PROGRAM MAIN
VAR
	bInit 	  : BOOL := FALSE; // flag for initialization
	bTaskDone : BOOL := FALSE;
END_VAR


// Command related
VAR
	fb_CommandProcess : FB_CommandProcess; // Process data from host and transfer data to Cpp
END_VAR
	
// Scope Server
VAR
	fb_GenerateFileSuffixByTime : FB_GenerateFileSuffixByTime; 	// Generate file suffix by system time
	fb_ScopeServer 		  		: FB_ScopeServer; 	  			// Record .svdx file
	bScopeRun 			  		: BOOL := FALSE; 		  		// Flag of starting or stoping scope server
	fb_ExportScopeData 	  		: FB_ExportScopeData;   		// Export recorded data after finishing 
	bExportData    		  		: BOOL := FALSE; 		  		// Flag of exporting data to file
END_VAR

// Initialize and Config load
VAR
	bBufferFilled 	 : BOOL := FALSE; // Flag reflects success or failure of initializing ring buffer
	bMcInfoLoaded 	 : BOOL := FALSE; // Flag reflects success or failure of loading motor info file
	bPanelInfoLoaded : BOOL := FALSE; // Flag reflects success or failure of loading panel info file
	fb_MotorInfoLoad : FB_MotorInfoLoad;
END_VAR

IF (NOT bInit) THEN
	
	bInit := mInitialize();
	
ELSE
	
	mInput();
	
	mOutput();
	
END_IF


// Scope Data Record
fb_ScopeServer(
	bExternalTriggerEvent	:= bScopeRun , 
	sConfigFile				:= GlobalVar.RECORD_CONFIG_PATH, 
	sSaveFile				:= CONCAT(GlobalVar.SAVE_SVDX_PREFIX, fb_GenerateFileSuffixByTime.SAVE_SVDX_SUFFIX));
	
fb_ExportScopeData(
	sNetId					:= '' , 
	bExport					:= bExportData , 
	svd						:= fb_ScopeServer.sSaveFile , 
	target					:= CONCAT(GlobalVar.SAVE_CSV_PREFIX, fb_GenerateFileSuffixByTime.SAVE_CSV_SUFFIX) , 
	config					:= GlobalVar.RECORD_CONFIG_XML_PATH);

METHOD mInitialize : BOOL
// Wait for the following initialization
// Step 1. Host Machine fills command buffer;
// Step 2. Current module finish loading MotionControl xml file;
// Step 3. Current module finish loading Panel xml file;
mInitialize := FALSE;

// Get time to generate suffix of files saved by scope server
fb_GenerateFileSuffixByTime();

// Step 1
IF NOT bBufferFilled THEN
	bBufferFilled := fb_CommandProcess.mInitialize();
END_IF


// Step 2 
IF NOT bMcInfoLoaded THEN
	fb_MotorInfoLoad();
	bMcInfoLoaded := fb_MotorInfoLoad.bExecuteSuccess;
END_IF


// Step 3
IF NOT bPanelInfoLoaded THEN
	bPanelInfoLoaded := TRUE;
END_IF

// Finish all initialization steps.
IF bBufferFilled AND bMcInfoLoaded AND bPanelInfoLoaded THEN
	
	// Start recording data
	bScopeRun := TRUE;
	
	// End initialization
	mInitialize := TRUE;
END_IF
END_METHOD

METHOD mInput : BOOL
VAR_INPUT
END_VAR
// Receive inputs from Hardware and other modules.
END_METHOD

METHOD mOutput : BOOL
VAR_INPUT
END_VAR
// Send outputs to Hardware and other modules.

mOutput := FALSE;

IF fb_CommandProcess.mSendCommand() THEN
	mOutput := TRUE;
ELSE
	// TODO: add judgment on whether the task is finished
	IF bTaskDone THEN
		bScopeRun := FALSE;
		
		// TODO: Add a delay between stop scope and start export
		// bExportData := TRUE;
	END_IF
	
	//RETURN;
	
END_IF
END_METHOD

END_PROGRAM

(* stored: Version 1.1.0.1
   POU MAIN: Id {65f328a0-4d74-4a01-8aa5-7e8c2290d3c3}, SpecialFunc None
   Method mInitialize: Id {9586f67e-0d90-4ec0-811a-a2c911cc73f9}
   Method mInput: Id {4779c18a-9e96-4364-9e93-c017388d8244}
   Method mOutput: Id {e076596c-b196-4e95-9e7b-70f2484e0f67} *)
